# EPICS substitutions: PIP-II/RFPI2/rfpi-fdr-sw-main-ioc/kriaApp/Db/reset.substitutions
file expert.template {
pattern{ acc, sys, group, num }
{ PIP2IT, pHB650, RFPI, kria }
{ PIP2IT, pHB650, RFPI, kria }
{ PIP2IT, pHB650, RFPI, kria }
{ PIP2IT, pHB650, RFPI, kria }
}
